// TwinCAT 3 PLC project plc
// ProgramVersion: 3.1.4026.21
// libraries:
//   Tc2_MC2, * (Beckhoff Automation GmbH)
//   Tc2_Standard, * (Beckhoff Automation GmbH)
//   Tc2_System, * (Beckhoff Automation GmbH)
// project tree:
//   GVLs/ GVL.TcGVL
//   / PlcTask.TcTTO
//   DUTs/ E_AxisState.TcDUT
//   POUs/ MAIN.TcPOU, FB_AxisControl.TcPOU
// real-time tasks:
//   TASK PlcTask: cycle T#10ms, priority 20, ADS port 350
// motion (NC):
//   TASK NC-Task 1 SAF: cycle T#2ms, priority 4, ADS port 501
//   TASK NC-Task 1 SVB: cycle T#10ms, priority 8, ADS port 511
//   AXIS Axis (id 1)
// variable links:
//   (this object) <-> NC-Task 1 SAF/Axes/Axis
//     PlcTask Inputs/GVL.ncAxis.NcToPlc <-> Outputs/ToPlc
//     PlcTask Outputs/GVL.ncAxis.PlcToNc <-> Inputs/FromPlc

CONFIGURATION plc
    RESOURCE PLC ON TwinCAT3
        TASK PlcTask(INTERVAL := T#10ms, PRIORITY := 20);
        PROGRAM MAIN WITH PlcTask : MAIN;
    END_RESOURCE
END_CONFIGURATION

// ---- DUTs/E_AxisState.TcDUT
{attribute 'qualified_only'}
(* States for the axis shuttle state machine in MAIN. *)
TYPE E_AxisState :
(
    eIDLE           :=  0,  // Axis unpowered, waiting for bStart
    ePOWERING_ON    := 10,  // Power enabled, waiting for axis ready
    eMOVE_TO_A      := 20,  // Issue move to position A
    eWAIT_MOVE_A    := 30,  // Waiting for move-to-A to complete
    eMOVE_TO_B      := 40,  // Issue move to position B
    eWAIT_MOVE_B    := 50,  // Waiting for move-to-B to complete
    eERROR          := 99   // Axis error — waiting for bReset
);
END_TYPE

// ---- GVLs/GVL.TcGVL
{attribute 'qualified_only'}
VAR_GLOBAL
    ncAxis          : AXIS_REF;         // Link to NC axis in the I/O tree
END_VAR

// ---- POUs/MAIN.TcPOU
PROGRAM MAIN
VAR
    (* ── Axis objects ─────────────────────────────────────────────────────── *)
    fbAxis          : FB_AxisControl;

    (* ── Operator commands (write from HMI / watch window) ───────────────── *)
    bStart          : BOOL;             // Rising edge — start shuttle sequence
    bStop           : BOOL;             // TRUE — stop sequence and power down
    bReset          : BOOL;             // Rising edge — reset axis error

    (* ── Shuttle parameters ───────────────────────────────────────────────── *)
    fPosA           : LREAL := 0.0;     // Position A [axis unit]
    fPosB           : LREAL := 100.0;   // Position B [axis unit]
    fVelocity       : LREAL := 50.0;    // Move velocity     [axis unit / s]
    fAcceleration   : LREAL := 500.0;   // Acceleration      [axis unit / s²]
    fDeceleration   : LREAL := 500.0;   // Deceleration      [axis unit / s²]
    fJerk           : LREAL := 0.0;     // Jerk limit (0 = disabled)

    (* ── State machine ────────────────────────────────────────────────────── *)
    eState          : E_AxisState := E_AxisState.eIDLE;

    (* ── Internal FB drive signals ───────────────────────────────────────── *)
    bEnableAxis     : BOOL;             // Drives fbAxis.bEnable every cycle
    bMoveCmd        : BOOL;             // Single-cycle rising edge for fbAxis.bMoveAbsolute
    fMoveTarget     : LREAL;            // Active target forwarded to fbAxis
END_VAR

// ── State machine ─────────────────────────────────────────────────────────────
CASE eState OF

    // ── eIDLE ──────────────────────────────────────────────────────────────
    // Axis is unpowered. Wait for the operator to press Start.
    E_AxisState.eIDLE:
        bEnableAxis := FALSE;
        IF bStart THEN
            bStart  := FALSE;   // consume the edge
            eState  := E_AxisState.ePOWERING_ON;
        END_IF

    // ── ePOWERING_ON ───────────────────────────────────────────────────────
    // Power is applied. Wait until the axis reports bReady (servo on, no error).
    E_AxisState.ePOWERING_ON:
        bEnableAxis := TRUE;
        IF fbAxis.bReady THEN
            eState := E_AxisState.eMOVE_TO_A;
        END_IF

    // ── eMOVE_TO_A ─────────────────────────────────────────────────────────
    // Assert bMoveCmd for exactly one PLC cycle to generate the rising edge
    // that triggers MC_MoveAbsolute toward position A, then advance immediately.
    E_AxisState.eMOVE_TO_A:
        fMoveTarget := fPosA;
        bMoveCmd    := TRUE;
        eState      := E_AxisState.eWAIT_MOVE_A;

    // ── eWAIT_MOVE_A ───────────────────────────────────────────────────────
    // bMoveCmd is cleared so MC_MoveAbsolute executes without re-triggering.
    // Proceed to B once the move is complete.
    E_AxisState.eWAIT_MOVE_A:
        bMoveCmd := FALSE;
        IF fbAxis.bMoveDone THEN
            eState := E_AxisState.eMOVE_TO_B;
        END_IF

    // ── eMOVE_TO_B ─────────────────────────────────────────────────────────
    E_AxisState.eMOVE_TO_B:
        fMoveTarget := fPosB;
        bMoveCmd    := TRUE;
        eState      := E_AxisState.eWAIT_MOVE_B;

    // ── eWAIT_MOVE_B ───────────────────────────────────────────────────────
    // Once position B is reached, loop back and head to A again.
    E_AxisState.eWAIT_MOVE_B:
        bMoveCmd := FALSE;
        IF fbAxis.bMoveDone THEN
            eState := E_AxisState.eMOVE_TO_A;
        END_IF

    // ── eERROR ─────────────────────────────────────────────────────────────
    // Power is removed. The operator must pulse bReset to clear the axis error.
    // FB_AxisControl forwards bReset to MC_Reset every cycle; once MC_Reset
    // reports Done the axis error is cleared and we return to eIDLE.
    E_AxisState.eERROR:
        bEnableAxis := FALSE;
        bMoveCmd    := FALSE;
        IF fbAxis.bResetDone THEN
            eState := E_AxisState.eIDLE;
        END_IF

END_CASE

// ── Global stop ────────────────────────────────────────────────────────────────
// Accepted from any active state; powers the axis down and returns to eIDLE.
IF bStop
    AND eState <> E_AxisState.eIDLE
    AND eState <> E_AxisState.eERROR
THEN
    bStop       := FALSE;
    bMoveCmd    := FALSE;
    bEnableAxis := FALSE;
    eState      := E_AxisState.eIDLE;
END_IF

// ── Error guard ────────────────────────────────────────────────────────────────
// Catch axis errors that surface during any active state.
IF fbAxis.bError
    AND eState <> E_AxisState.eERROR
    AND eState <> E_AxisState.eIDLE
THEN
    bMoveCmd    := FALSE;
    bEnableAxis := FALSE;
    eState      := E_AxisState.eERROR;
END_IF

// ── Call FB_AxisControl ────────────────────────────────────────────────────────
// Must be the last statement so that bMoveCmd and bEnableAxis reflect the
// decisions taken in this cycle before being forwarded to the MC FBs.
fbAxis(
    stAxis          := GVL.ncAxis,
    bEnable         := bEnableAxis,
    bEnablePositive := bEnableAxis,
    bEnableNegative := bEnableAxis,
    bReset          := bReset,
    bMoveAbsolute   := bMoveCmd,
    fTargetPosition := fMoveTarget,
    fVelocity       := fVelocity,
    fAcceleration   := fAcceleration,
    fDeceleration   := fDeceleration,
    fJerk           := fJerk
);

END_PROGRAM

// ---- POUs/FB_AxisControl.TcPOU
{attribute 'reflection'}
(* ============================================================
   FB_AxisControl
   Purpose : Wraps the core Tc2_MC2 motion function blocks for
             a single NC axis — power, reset and absolute move.
   Requires: Tc2_MC2 library reference in the PLC project.
   Usage   : Call this FB every PLC cycle. Drive inputs with
             rising-edge signals from your HMI / state machine.
   ============================================================ *)
FUNCTION_BLOCK FB_AxisControl
VAR_IN_OUT
    (* NC axis reference — link to the axis object in the I/O tree. *)
    stAxis              : AXIS_REF;
END_VAR
VAR_INPUT
    (* --- Power control --- *)
    bEnable             : BOOL;     // TRUE = servo on (MC_Power Enable)
    bEnablePositive     : BOOL;     // TRUE = allow motion in positive direction
    bEnableNegative     : BOOL;     // TRUE = allow motion in negative direction

    (* --- Reset --- *)
    bReset              : BOOL;     // Rising edge clears axis error and re-enables

    (* --- Absolute move --- *)
    bMoveAbsolute       : BOOL;     // Rising edge starts absolute positioning move
    fTargetPosition     : LREAL;    // Target position [axis unit]
    fVelocity           : LREAL;    // Move velocity    [axis unit / s]
    fAcceleration       : LREAL;    // Acceleration     [axis unit / s²]
    fDeceleration       : LREAL;    // Deceleration     [axis unit / s²]
    fJerk               : LREAL;    // Jerk limit       [axis unit / s³], 0 = disabled
END_VAR
VAR_OUTPUT
    (* --- Axis status feedback --- *)
    bPowered            : BOOL;     // Axis servo is on (MC_Power.Status)
    bReady              : BOOL;     // Powered and no error — ready for commands
    bBusy               : BOOL;     // Any motion command is currently active

    (* --- MC_Reset feedback --- *)
    bResetDone          : BOOL;     // Reset completed successfully
    bResetBusy          : BOOL;     // Reset in progress
    bResetError         : BOOL;     // Reset FB error
    nResetErrorId       : UDINT;    // Reset ADS error ID

    (* --- MC_MoveAbsolute feedback --- *)
    bMoveDone           : BOOL;     // Absolute move reached target position
    bMoveBusy           : BOOL;     // Absolute move in progress
    bMoveActive         : BOOL;     // Absolute move command is active on the axis
    bMoveError          : BOOL;     // Absolute move FB error
    nMoveErrorId        : UDINT;    // Absolute move ADS error ID

    (* --- Aggregated error --- *)
    bError              : BOOL;     // Any of the motion FBs has an active error
    nErrorId            : UDINT;    // First non-zero error ID among all FBs

    (* --- Live axis data --- *)
    fActPosition        : LREAL;    // Actual position [axis unit]
    fActVelocity        : LREAL;    // Actual velocity [axis unit / s]
END_VAR
VAR
    fbMcPower           : MC_Power;
    fbMcReset           : MC_Reset;
    fbMcMoveAbsolute    : MC_MoveAbsolute;
END_VAR

// Get axis status
stAxis.ReadStatus();

// ── MC_Power ──────────────────────────────────────────────────────────────────
// Continuously driven every cycle; axis stays powered as long as bEnable = TRUE.
fbMcPower(
    Axis            := stAxis,
    Enable          := bEnable,
    Enable_Positive := bEnablePositive,
    Enable_Negative := bEnableNegative,
    Override        := 100.0,           // velocity override 100 %
    BufferMode      := MC_Aborting
);
bPowered := fbMcPower.Status;

// ── MC_Reset ──────────────────────────────────────────────────────────────────
// Triggered by a rising edge on bReset; clears axis errors so MC_Power can
// re-establish servo state.
fbMcReset(
    Axis    := stAxis,
    Execute := bReset
);
bResetDone    := fbMcReset.Done;
bResetBusy    := fbMcReset.Busy;
bResetError   := fbMcReset.Error;
nResetErrorId := fbMcReset.ErrorID;

// ── MC_MoveAbsolute ───────────────────────────────────────────────────────────
// Triggered by a rising edge on bMoveAbsolute. The axis must be powered and
// error-free before issuing the command.
fbMcMoveAbsolute(
    Axis         := GVL.ncAxis,
    Execute      := bMoveAbsolute,
    Position     := fTargetPosition,
    Velocity     := fVelocity,
    Acceleration := fAcceleration,
    Deceleration := fDeceleration,
    Jerk         := fJerk,
    BufferMode   := MC_Aborting
);
bMoveDone    := fbMcMoveAbsolute.Done;
bMoveBusy    := fbMcMoveAbsolute.Busy;
bMoveActive  := fbMcMoveAbsolute.Active;
bMoveError   := fbMcMoveAbsolute.Error;
nMoveErrorId := fbMcMoveAbsolute.ErrorID;

// ── Aggregated status ─────────────────────────────────────────────────────────
bBusy  := bResetBusy OR bMoveBusy;
bError := fbMcPower.Error OR bResetError OR bMoveError;

// Expose the first non-zero error ID for quick diagnostics.
IF fbMcPower.Error THEN
    nErrorId := fbMcPower.ErrorID;
ELSIF bResetError THEN
    nErrorId := nResetErrorId;
ELSIF bMoveError THEN
    nErrorId := nMoveErrorId;
ELSE
    nErrorId := 0;
END_IF

// Axis is truly ready only when powered and no error is present.
bReady := bPowered AND NOT bError;

// ── Live axis position and velocity ───────────────────────────────────────────
// Read directly from the AXIS_REF NcToPlc structure (updated by the NC task).
fActPosition := stAxis.NcToPlc.ActPos;
fActVelocity := stAxis.NcToPlc.ActVelo;

END_FUNCTION_BLOCK
